TYPE PositionStatus :
STRUCT
	Busy : BOOL;
	InTarget : BOOL;
	Warning : BOOL;
	Error : BOOL;
	Calibrated : BOOL;
	Accelerate : BOOL;
	Decelerate : BOOL;
	ReadyToExecute : BOOL;
END_STRUCT
END_TYPE

(* stored: Version 1.1.0.1, ProductVersion 3.1.4024.11
   DUT PositionStatus: Id {e3ea44e7-ca90-449e-8ae8-fc25113275c4} *)
